ABB RAPID module: ROS_motion_right.mod

MODULE ROS_motion_right

! Software License Agreement (BSD License)
!
! Copyright (c) 2012, Edward Venator, Case Western Reserve University
! Copyright (c) 2012, Jeremy Zoss, Southwest Research Institute
! All rights reserved.
!
! Redistribution and use in source and binary forms, with or without modification,
! are permitted provided that the following conditions are met:
!
!   Redistributions of source code must retain the above copyright notice, this
!       list of conditions and the following disclaimer.
!   Redistributions in binary form must reproduce the above copyright notice, this
!       list of conditions and the following disclaimer in the documentation
!       and/or other materials provided with the distribution.
!   Neither the name of the Case Western Reserve University nor the names of its contributors
!       may be used to endorse or promote products derived from this software without
!       specific prior written permission.
!
! THIS SOFTWARE IS PROVIDED BY THE COPYRIGHT HOLDERS AND CONTRIBUTORS "AS IS" AND ANY
! EXPRESS OR IMPLIED WARRANTIES, INCLUDING, BUT NOT LIMITED TO, THE IMPLIED WARRANTIES
! OF MERCHANTABILITY AND FITNESS FOR A PARTICULAR PURPOSE ARE DISCLAIMED. IN NO EVENT
! SHALL THE COPYRIGHT HOLDER OR CONTRIBUTORS BE LIABLE FOR ANY DIRECT, INDIRECT,
! INCIDENTAL, SPECIAL, EXEMPLARY, OR CONSEQUENTIAL DAMAGES (INCLUDING, BUT NOT LIMITED
! TO, PROCUREMENT OF SUBSTITUTE GOODS OR SERVICES; LOSS OF USE, DATA, OR PROFITS; OR
! BUSINESS INTERRUPTION) HOWEVER CAUSED AND ON ANY THEORY OF LIABILITY, WHETHER IN
! CONTRACT, STRICT LIABILITY, OR TORT (INCLUDING NEGLIGENCE OR OTHERWISE) ARISING IN ANY
! WAY OUT OF THE USE OF THIS SOFTWARE, EVEN IF ADVISED OF THE POSSIBILITY OF SUCH DAMAGE.

LOCAL CONST zonedata DEFAULT_CORNER_DIST := z10;
LOCAL VAR ROS_joint_trajectory_pt trajectory{MAX_TRAJ_LENGTH};
LOCAL VAR num trajectory_size := 0;
LOCAL VAR intnum intr_new_trajectory;
LOCAL CONST jointtarget jpos_Cal_Home_R:=[[0,-130,30,0,40,0],[-135,9E+09,9E+09,9E+09,9E+09,9E+09]];
LOCAL CONST robtarget Target_Cal_Home_R:=[[-5.94,-184.30,200.00],[0.0637387,-0.840372,-0.106584,-0.527591],[0,0,0,4],[-101.793,9E+09,9E+09,9E+09,9E+09,9E+09]];

PROC main()
    VAR num current_index;
    VAR jointtarget target;
    VAR speeddata move_speed := v10;  ! default speed
    VAR zonedata stop_mode;
    VAR bool skip_move;

    ! Set up interrupt to watch for new trajectory
    IDelete intr_new_trajectory;    ! clear interrupt handler, in case restarted with ExitCycle
    CONNECT intr_new_trajectory WITH new_trajectory_handler;
    IPers ROS_new_trajectory_right, intr_new_trajectory;

    ! Move the right arm to the Calibration Home position, modified by honghao
    MoveAbsJ jpos_Cal_Home_R,v100,z5,tool0\WObj:=wobj0;
    WaitTime 2;

    WHILE true DO
        ! Check for new Trajectory
        IF (ROS_new_trajectory_right)
            init_trajectory;

        ! execute all points in this trajectory
        IF (trajectory_size > 0) THEN
            FOR current_index FROM 1 TO trajectory_size DO
                target.robax := trajectory{current_index}.joint_pos.robax;
                target.extax.eax_a := trajectory{current_index}.joint_pos.extax.eax_a;

                skip_move := (current_index = 1) AND is_near(target.robax, 0.1);

                stop_mode := DEFAULT_CORNER_DIST;  ! assume we're smoothing between points
                IF (current_index = trajectory_size) stop_mode := fine;  ! stop at path end

                ! Execute move command
                IF (NOT skip_move)
                    MoveAbsJ target, move_speed, \T:=trajectory{current_index}.duration, stop_mode, tool0;
            ENDFOR

            trajectory_size := 0;  ! trajectory done
        ENDIF

        WaitTime 0.05;  ! Throttle loop while waiting for new command
    ENDWHILE
ERROR
    ErrWrite \W, "Motion Error", "Error executing motion.  Aborting trajectory.";
    abort_trajectory;
ENDPROC

LOCAL PROC init_trajectory()
    clear_path;                    ! cancel any active motions

    WaitTestAndSet ROS_trajectory_lock_right;  ! acquire data-lock
      trajectory := ROS_trajectory_right;            ! copy to local var
      trajectory_size := ROS_trajectory_size_right;  ! copy to local var
      ROS_new_trajectory_right := FALSE;
    ROS_trajectory_lock_right := FALSE;         ! release data-lock
ENDPROC

LOCAL FUNC bool is_near(robjoint target, num tol)
    VAR jointtarget curr_jnt;

    curr_jnt := CJointT();

    RETURN ( ABS(curr_jnt.robax.rax_1 - target.rax_1) < tol )
       AND ( ABS(curr_jnt.robax.rax_2 - target.rax_2) < tol )
       AND ( ABS(curr_jnt.robax.rax_3 - target.rax_3) < tol )
       AND ( ABS(curr_jnt.robax.rax_4 - target.rax_4) < tol )
       AND ( ABS(curr_jnt.robax.rax_5 - target.rax_5) < tol )
       AND ( ABS(curr_jnt.robax.rax_6 - target.rax_6) < tol );
ENDFUNC

LOCAL PROC abort_trajectory()
    trajectory_size := 0;  ! "clear" local trajectory
    clear_path;
    ExitCycle;  ! restart program
ENDPROC

LOCAL PROC clear_path()
    IF ( NOT (IsStopMoveAct(\FromMoveTask) OR IsStopMoveAct(\FromNonMoveTask)) )
        StopMove;          ! stop any active motions
    ClearPath;             ! clear queued motion commands
    StartMove;             ! re-enable motions
ENDPROC

LOCAL TRAP new_trajectory_handler
    IF (NOT ROS_new_trajectory_right) RETURN;

    abort_trajectory;
ENDTRAP

ENDMODULE
